KUKA KRL program: FOLLOWSHAPE.src, FOLLOWSHAPE.dat

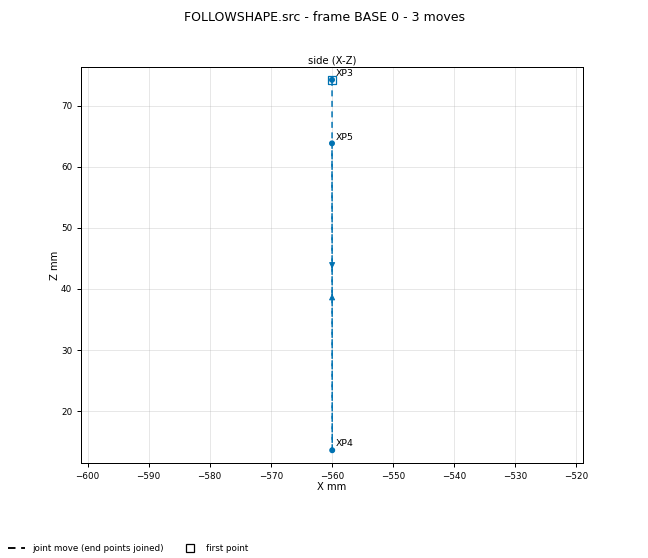
[picture p0: tool path of FOLLOWSHAPE.src in frame BASE 0, 3 of 3 moves have a stored position in this frame; points joined in program order, loops and branches not executed]
--- FOLLOWSHAPE.src ---
&ACCESS RVP
&REL 80
&PARAM TEMPLATE = C:\KRC\Roboter\Template\vorgabe
&PARAM EDITMASK = *
DEF FOLLOWSHAPE( )

DECL BOOL TEMP
DECL BOOL HEMP
DECL TORQUE_TCP_EST MyTorque
;FOLD INI
  ;FOLD BASISTECH INI
    GLOBAL INTERRUPT DECL 3 WHEN $STOPMESS==TRUE DO IR_STOPM ( )
    INTERRUPT ON 3
    BAS (#INITMOV,0 )
  ;ENDFOLD (BASISTECH INI)
  ;FOLD USER INI
    ;Make your modifications here
LOGROBOTDATA=TRUE
SERVERCONNECTED=TRUE
TCPCONNECTION=FALSE
  ;ENDFOLD (USER INI)
;ENDFOLD (INI)

$STIFFNESS.STRATEGY=10
$STIFFNESS.COMMIT=TRUE

;FOLD PTP P3 Vel=100 % PDAT3 Tool[5]:Pneumatic_gripper_probe Base[0];%{PE}%R 5.6.11,%MKUKATPBASIS,%CMOVE,%VPTP,%P 1:PTP, 2:P3, 3:, 5:100, 7:PDAT3
$BWDSTART=FALSE
PDAT_ACT=PPDAT3
FDAT_ACT=FP3
BAS(#PTP_PARAMS,100)
PTP XP3
;ENDFOLD

;FOLD PTP P4 Vel=100 % PDAT4 Tool[5]:Pneumatic_gripper_probe Base[0];%{PE}%R 5.6.11,%MKUKATPBASIS,%CMOVE,%VPTP,%P 1:PTP, 2:P4, 3:, 5:100, 7:PDAT4
$BWDSTART=FALSE
PDAT_ACT=PPDAT4
FDAT_ACT=FP4
BAS(#PTP_PARAMS,100)
PTP XP4
;ENDFOLD

$OV_PRO=10

TEMP=TRIGFORCE()

HEMP=TRIGBACK()


$STIFFNESS.STRATEGY=10
$STIFFNESS.COMMIT=TRUE

$OV_PRO=100


;FOLD PTP P5 Vel=100 % PDAT5 Tool[5]:Pneumatic_gripper_probe Base[0];%{PE}%R 5.6.11,%MKUKATPBASIS,%CMOVE,%VPTP,%P 1:PTP, 2:P5, 3:, 5:100, 7:PDAT5
$BWDSTART=FALSE
PDAT_ACT=PPDAT5
FDAT_ACT=FP5
BAS(#PTP_PARAMS,100)
PTP XP5
;ENDFOLD

LOGROBOTDATA=FALSE
SERVERCONNECTED=FALSE
TCPCONNECTION=FALSE

END

--- FOLLOWSHAPE.dat ---
&ACCESS RVP
&REL 80
&PARAM TEMPLATE = C:\KRC\Roboter\Template\vorgabe
&PARAM EDITMASK = *
DEFDAT  FOLLOWSHAPE
;FOLD EXTERNAL DECLARATIONS;%{PE}%MKUKATPBASIS,%CEXT,%VCOMMON,%P
;FOLD BASISTECH EXT;%{PE}%MKUKATPBASIS,%CEXT,%VEXT,%P
EXT  BAS (BAS_COMMAND  :IN,REAL  :IN )
DECL INT SUCCESS
;ENDFOLD (BASISTECH EXT)
;FOLD USER EXT;%{E}%MKUKATPUSER,%CEXT,%VEXT,%P
;Make here your modifications

;ENDFOLD (USER EXT)
;ENDFOLD (EXTERNAL DECLARATIONS)
DECL BASIS_SUGG_T LAST_BASIS={POINT1[] "P5                      ",POINT2[] "P5                      ",CP_PARAMS[] "CPDAT0                  ",PTP_PARAMS[] "PDAT5                   ",CONT[] "                        ",CP_VEL[] "2.0                     ",PTP_VEL[] "100                     ",SYNC_PARAMS[] "SYNCDAT                 ",SPL_NAME[] "S0                      "}
DECL INT LAST_XP_POINT=4
DECL E6POS XP1={X -559.978577,Y -436.973907,Z 74.2913437,A 89.9966125,B -0.00364325289,C 179.994705,S 1,T 12,E1 0.252170593,E2 0.0,E3 0.0,E4 0.0,E5 0.0,E6 0.0}
DECL FDAT FP1={TOOL_NO 5,BASE_NO 0,IPO_FRAME #BASE,POINT2[] " ",TQ_STATE FALSE}
DECL PDAT PPDAT1={VEL 100.0,ACC 100.0,APO_DIST 100.0,APO_MODE #CPTP}
DECL E6POS XP2={X -559.978577,Y -436.973907,Z 74.2913437,A 89.9966125,B -0.00364325289,C 179.994705,S 1,T 12,E1 0.252170593,E2 0.0,E3 0.0,E4 0.0,E5 0.0,E6 0.0}
DECL FDAT FP2={TOOL_NO 5,BASE_NO 0,IPO_FRAME #BASE,POINT2[] " ",TQ_STATE FALSE}
DECL PDAT PPDAT2={VEL 100.0,ACC 100.0,APO_DIST 100.0,APO_MODE #CPTP}
DECL E6POS XP3={X -559.963013,Y -436.935089,Z 74.2567368,A 89.990799,B -0.00836852286,C 179.989594,S 1,T 12,E1 0.250994712,E2 0.0,E3 0.0,E4 0.0,E5 0.0,E6 0.0}
DECL FDAT FP3={TOOL_NO 5,BASE_NO 0,IPO_FRAME #BASE,POINT2[] " ",TQ_STATE FALSE}
DECL PDAT PPDAT3={VEL 100.0,ACC 100.0,APO_DIST 100.0,APO_MODE #CPTP}
DECL E6POS XP4={X -559.933594,Y -436.914215,Z 13.5857201,A 89.9906006,B -0.01245772,C 179.984604,S 1,T 12,E1 0.250702888,E2 0.0,E3 0.0,E4 0.0,E5 0.0,E6 0.0}
DECL FDAT FP4={TOOL_NO 5,BASE_NO 0,IPO_FRAME #BASE,POINT2[] " ",TQ_STATE FALSE}
DECL PDAT PPDAT4={VEL 100.0,ACC 100.0,APO_DIST 100.0,APO_MODE #CPTP}
DECL E6POS XP5={X -559.970215,Y -436.928406,Z 63.8572617,A 89.9841385,B -0.00853981823,C 179.990494,S 1,T 12,E1 0.250556886,E2 0.0,E3 0.0,E4 0.0,E5 0.0,E6 0.0}
DECL FDAT FP5={TOOL_NO 5,BASE_NO 0,IPO_FRAME #BASE,POINT2[] " ",TQ_STATE FALSE}
DECL PDAT PPDAT5={VEL 100.0,ACC 100.0,APO_DIST 100.0,APO_MODE #CPTP}
ENDDAT
